{attribute 'qualified_only'}
//{attribute 'strict'}
{attribute 'to_string'}
TYPE E_LIST_STATE :
(
  LIST_STATE_INVALID,
	LIST_STATE_NULL,
  LIST_STATE_INIT      := 10,
  LIST_STATE_GET_HEAD  := 20,
  LIST_STATE_GET_TAIL  := 30,
  LIST_STATE_ADD_HEAD  := 40,
  LIST_STATE_ADD_TAIL  := 50,
  LIST_STATE_DEL_HEAD  := 60,
  LIST_STATE_DEL_TAIL  := 70
)UINT;
END_TYPE

(* stored: Version 1.1.0.1, ProductVersion 3.1.4026.18
   DUT E_LIST_STATE: Id {4411f1d2-43b4-4333-b9da-04da929861fd} *)
